PROGRAM PRG_CML_ValidationAsConfirmation
VAR

	rtrigNewOuterArrived				: R_TRIG;
	bNewOuterIsProccesing				: BOOL;
	tonValidationTimout					: TON;
	tofValidationTimout					: TOF;
	ftrigValidationTimout				: F_TRIG;
	bValidationTimeout					: BOOL;
	bValidationTimeoutReset				: BOOL;
	fbTooCloseCounter					: CTU;
	fbTimeoutCounter					: CTU;
	nCountTimeout					: WORD;
	nCountTooClose					: WORD;

	fbMasterListCamera				: FB_SCANNER_CameraSelect;
	(*stMasterListCameraOptions		: ST_SCANNER_Options := (eScannerType := E_MV_420_FULL, nImageBuffer := 1, nExpectedResp := 2);*)

	fbOuterValidationEvaluation		: FB_SCANNER_Evaluation;
	fbCheckForDuplicateMasterList	: FB_OUTER_CheckDuplicateStatus;

	rtrigOuterCameraDone				: R_TRIG;
	bOuterCameraDone				: BOOL;
	bDataReadyForValidation			: BOOL;
	bQAReject								: BOOL;

	sLastImageLableString				: T_OUTER_Barcode;

	fbPerformance							: FB_Interval;
	fbMoveOuterData						: FB_OUTER_MoveOuterStatus;
	fbCompleteDataFromConfirmation	: FB_OUTER_CompleteDataFromDB_SingleCam;
	fbMETSValidateOuterForReject			: FB_OUTER_ValidateOuterForReject;
	tofValidateOuterDoneForHMI			: TOF;
	fbMasterListUpdate					: FB_OUTER_MasterListUpdate;

	fbOuterLevelCounter				: FB_KPI_OuterLevelCounter;

	stLastOuterCompleted				: ST_OUTER_Status;
	sLastReadOuterBarcode			: T_OUTER_Barcode;
	sLastReadConfPackCode1			: T_PACK_Barcode;
	nOutersCompleted					: UDINT;
	bDoneInfo							: BOOL;
	rsTwoOutersOnRejectConv		: RS;
	bTwoOutersOnRejectConv			: BOOL;
	bCMLBiuldBackRejectActive		: BOOL;

	rtrigSetOuterValidationOK			: R_TRIG;
	rtrigSetOuterValidationNOK		: R_TRIG;
	rtrigResetValidationStatus			: R_TRIG;

	rsOuterRejectStation 				: RS;

	sRejectCode						: STRING(255);
	fbArchiveInvalidOuters			: FB_OUTER_ArchiveInvalidOuters;
	aReasonForReject					: ARRAY[0..50] OF STRING(255);
	bClearList							: BOOL;

	fbOuterProduced					: FB_KPI_GenericEfficiency;
	fbOuterInspection					: FB_KPI_OutersEfficiency;

	fbQARejectCounter				: FB_CTU32;
	fbOuterValidationIndexOK			: FB_CTU32;

	ctuConsecutiveOuterRejects		: CTU;
	nActualCount						: WORD;
END_VAR
VAR // added by the converter: edge detectors and wires of the graphical bodies
    _w1, _w2 : BOOL;
END_VAR

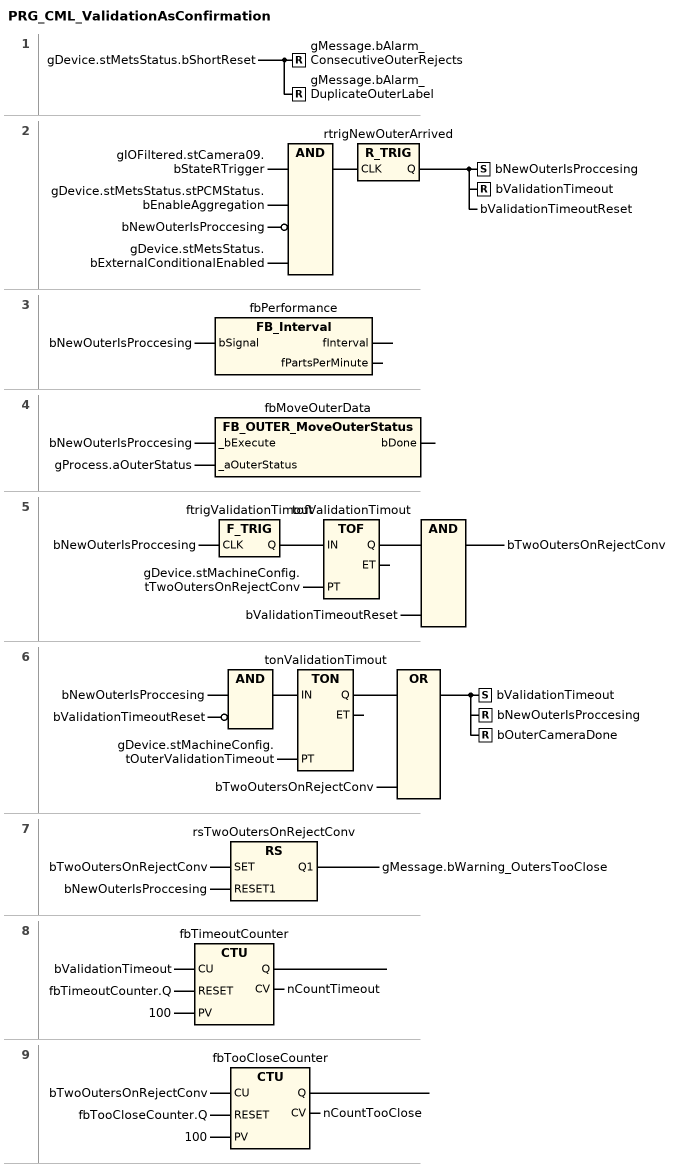
// NETWORK 1
gMessage.bAlarm_ConsecutiveOuterRejects R= gDevice.stMetsStatus.bShortReset;
gMessage.bAlarm_DuplicateOuterLabel R= gDevice.stMetsStatus.bShortReset;

// NETWORK 2
rtrigNewOuterArrived(CLK := gIOFiltered.stCamera09.bStateRTrigger AND gDevice.stMetsStatus.stPCMStatus.bEnableAggregation AND NOT bNewOuterIsProccesing AND gDevice.stMetsStatus.bExternalConditionalEnabled); // R_TRIG
bNewOuterIsProccesing S= rtrigNewOuterArrived.Q;
bValidationTimeout R= rtrigNewOuterArrived.Q;
bValidationTimeoutReset := rtrigNewOuterArrived.Q;

// NETWORK 3
fbPerformance(bSignal := bNewOuterIsProccesing); // FB_Interval

// NETWORK 4
fbMoveOuterData(_bExecute := bNewOuterIsProccesing, _aOuterStatus := gProcess.aOuterStatus); // FB_OUTER_MoveOuterStatus

// NETWORK 5
ftrigValidationTimout(CLK := bNewOuterIsProccesing); // F_TRIG
tofValidationTimout(IN := ftrigValidationTimout.Q, PT := gDevice.stMachineConfig.tTwoOutersOnRejectConv); // TOF
bTwoOutersOnRejectConv := tofValidationTimout.Q AND bValidationTimeoutReset;

// NETWORK 6
tonValidationTimout(IN := bNewOuterIsProccesing AND NOT bValidationTimeoutReset, PT := gDevice.stMachineConfig.tOuterValidationTimeout); // TON
_w1 := tonValidationTimout.Q OR bTwoOutersOnRejectConv;
bValidationTimeout S= _w1;
bNewOuterIsProccesing R= _w1;
bOuterCameraDone R= _w1;

// NETWORK 7
rsTwoOutersOnRejectConv(SET := bTwoOutersOnRejectConv, RESET1 := bNewOuterIsProccesing); // RS
gMessage.bWarning_OutersTooClose := rsTwoOutersOnRejectConv.Q1;

// NETWORK 8
fbTimeoutCounter(CU := bValidationTimeout, RESET := fbTimeoutCounter.Q, PV := 100, CV => nCountTimeout); // CTU

// NETWORK 9
fbTooCloseCounter(
    CU := bTwoOutersOnRejectConv,
    RESET := fbTooCloseCounter.Q,
    PV := 100,
    CV => nCountTooClose); // CTU

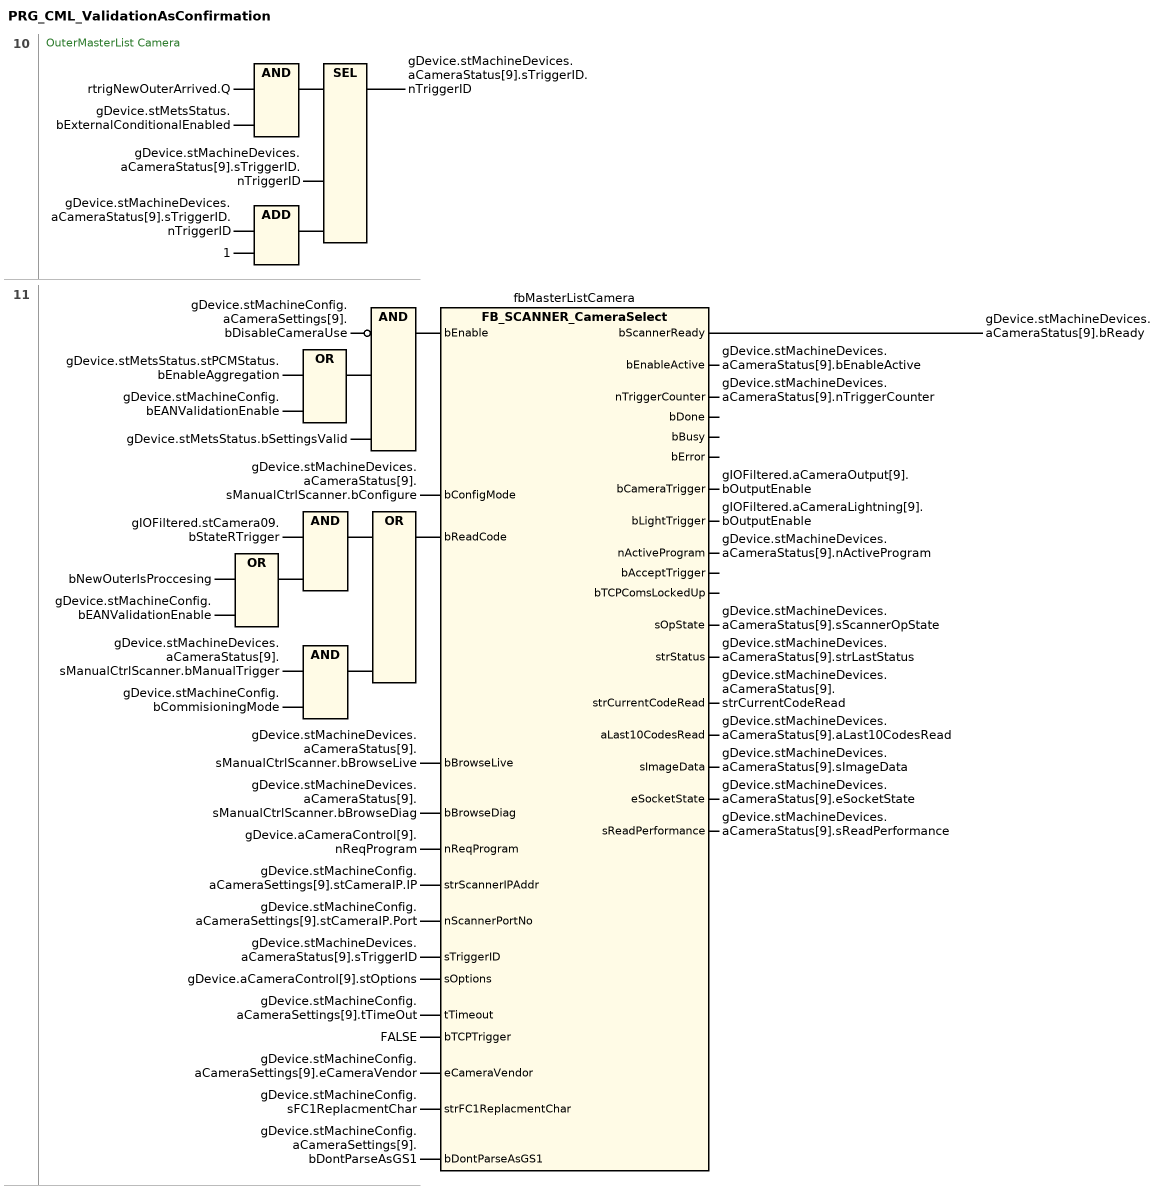
// NETWORK 10
// OuterMasterList Camera
gDevice.stMachineDevices.aCameraStatus[9].sTriggerID.nTriggerID := SEL(rtrigNewOuterArrived.Q AND gDevice.stMetsStatus.bExternalConditionalEnabled, gDevice.stMachineDevices.aCameraStatus[9].sTriggerID.nTriggerID, gDevice.stMachineDevices.aCameraStatus[9].sTriggerID.nTriggerID + 1);

// NETWORK 11
fbMasterListCamera(
    bEnable := NOT gDevice.stMachineConfig.aCameraSettings[9].bDisableCameraUse AND (gDevice.stMetsStatus.stPCMStatus.bEnableAggregation OR gDevice.stMachineConfig.bEANValidationEnable) AND gDevice.stMetsStatus.bSettingsValid,
    bConfigMode := gDevice.stMachineDevices.aCameraStatus[9].sManualCtrlScanner.bConfigure,
    bReadCode := gIOFiltered.stCamera09.bStateRTrigger AND (bNewOuterIsProccesing OR gDevice.stMachineConfig.bEANValidationEnable) OR gDevice.stMachineDevices.aCameraStatus[9].sManualCtrlScanner.bManualTrigger AND gDevice.stMachineConfig.bCommisioningMode,
    bBrowseLive := gDevice.stMachineDevices.aCameraStatus[9].sManualCtrlScanner.bBrowseLive,
    bBrowseDiag := gDevice.stMachineDevices.aCameraStatus[9].sManualCtrlScanner.bBrowseDiag,
    nReqProgram := gDevice.aCameraControl[9].nReqProgram,
    strScannerIPAddr := gDevice.stMachineConfig.aCameraSettings[9].stCameraIP.IP,
    nScannerPortNo := gDevice.stMachineConfig.aCameraSettings[9].stCameraIP.Port,
    sTriggerID := gDevice.stMachineDevices.aCameraStatus[9].sTriggerID,
    sOptions := gDevice.aCameraControl[9].stOptions,
    tTimeout := gDevice.stMachineConfig.aCameraSettings[9].tTimeOut,
    bTCPTrigger := FALSE,
    eCameraVendor := gDevice.stMachineConfig.aCameraSettings[9].eCameraVendor,
    strFC1ReplacmentChar := gDevice.stMachineConfig.sFC1ReplacmentChar,
    bDontParseAsGS1 := gDevice.stMachineConfig.aCameraSettings[9].bDontParseAsGS1,
    bEnableActive => gDevice.stMachineDevices.aCameraStatus[9].bEnableActive,
    nTriggerCounter => gDevice.stMachineDevices.aCameraStatus[9].nTriggerCounter,
    bCameraTrigger => gIOFiltered.aCameraOutput[9].bOutputEnable,
    bLightTrigger => gIOFiltered.aCameraLightning[9].bOutputEnable,
    nActiveProgram => gDevice.stMachineDevices.aCameraStatus[9].nActiveProgram,
    sOpState => gDevice.stMachineDevices.aCameraStatus[9].sScannerOpState,
    strStatus => gDevice.stMachineDevices.aCameraStatus[9].strLastStatus,
    strCurrentCodeRead => gDevice.stMachineDevices.aCameraStatus[9].strCurrentCodeRead,
    aLast10CodesRead => gDevice.stMachineDevices.aCameraStatus[9].aLast10CodesRead,
    sImageData => gDevice.stMachineDevices.aCameraStatus[9].sImageData,
    eSocketState => gDevice.stMachineDevices.aCameraStatus[9].eSocketState,
    sReadPerformance => gDevice.stMachineDevices.aCameraStatus[9].sReadPerformance); // FB_SCANNER_CameraSelect
gDevice.stMachineDevices.aCameraStatus[9].bReady := fbMasterListCamera.bScannerReady;

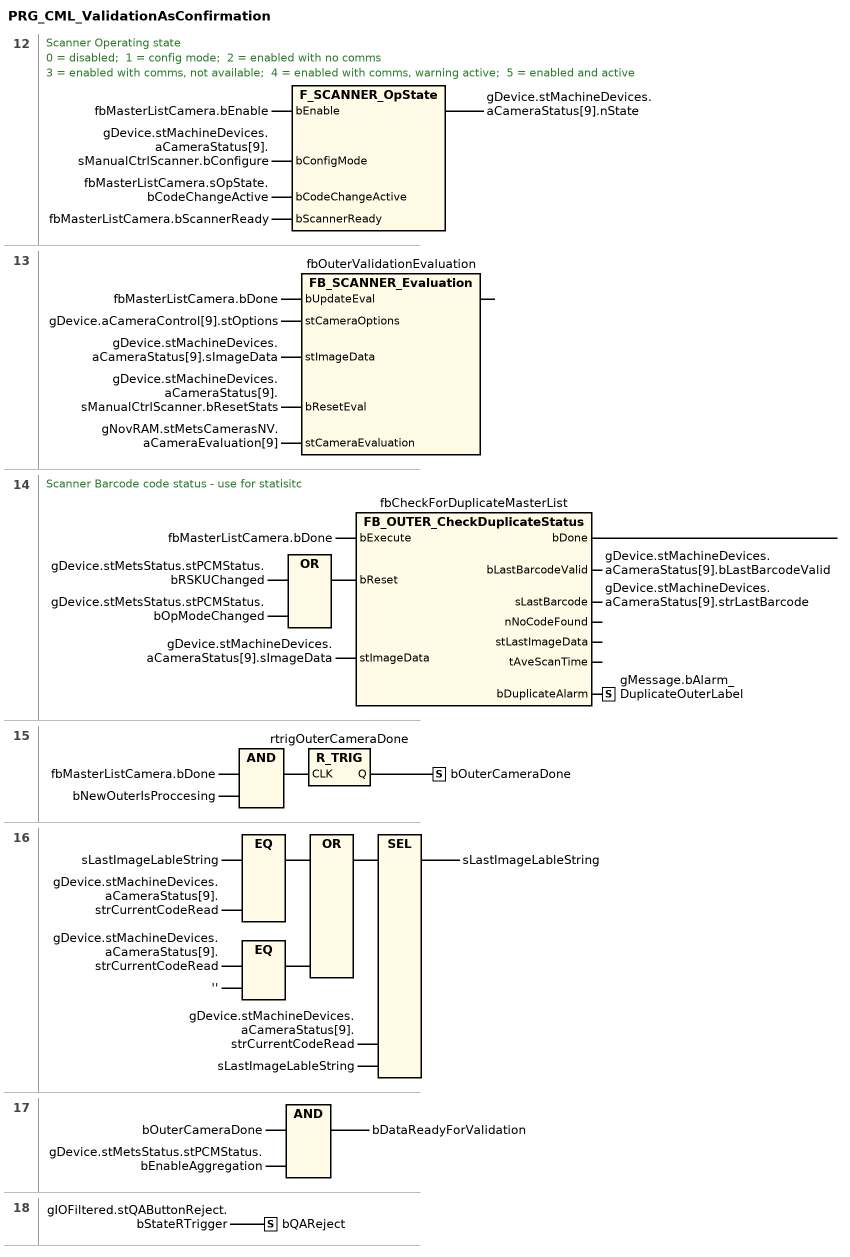
// NETWORK 12
// 					Scanner Operating state
// 0 = disabled;  1 = config mode;  2 = enabled with no comms
// 3 = enabled with comms, not available;  4 = enabled with comms, warning active;  5 = enabled and active
//
gDevice.stMachineDevices.aCameraStatus[9].nState := F_SCANNER_OpState(bEnable := fbMasterListCamera.bEnable, bConfigMode := gDevice.stMachineDevices.aCameraStatus[9].sManualCtrlScanner.bConfigure, bCodeChangeActive := fbMasterListCamera.sOpState.bCodeChangeActive, bScannerReady := fbMasterListCamera.bScannerReady);

// NETWORK 13
fbOuterValidationEvaluation(
    bUpdateEval := fbMasterListCamera.bDone,
    stCameraOptions := gDevice.aCameraControl[9].stOptions,
    stImageData := gDevice.stMachineDevices.aCameraStatus[9].sImageData,
    bResetEval := gDevice.stMachineDevices.aCameraStatus[9].sManualCtrlScanner.bResetStats,
    stCameraEvaluation := gNovRAM.stMetsCamerasNV.aCameraEvaluation[9]); // FB_SCANNER_Evaluation

// NETWORK 14
// Scanner Barcode code status - use for statisitc
fbCheckForDuplicateMasterList(
    bExecute := fbMasterListCamera.bDone,
    bReset := gDevice.stMetsStatus.stPCMStatus.bRSKUChanged OR gDevice.stMetsStatus.stPCMStatus.bOpModeChanged,
    stImageData := gDevice.stMachineDevices.aCameraStatus[9].sImageData,
    bLastBarcodeValid => gDevice.stMachineDevices.aCameraStatus[9].bLastBarcodeValid,
    sLastBarcode => gDevice.stMachineDevices.aCameraStatus[9].strLastBarcode); // FB_OUTER_CheckDuplicateStatus
gMessage.bAlarm_DuplicateOuterLabel S= fbCheckForDuplicateMasterList.bDuplicateAlarm;

// NETWORK 15
rtrigOuterCameraDone(CLK := fbMasterListCamera.bDone AND bNewOuterIsProccesing); // R_TRIG
bOuterCameraDone S= rtrigOuterCameraDone.Q;

// NETWORK 16
sLastImageLableString := SEL(sLastImageLableString = gDevice.stMachineDevices.aCameraStatus[9].strCurrentCodeRead OR gDevice.stMachineDevices.aCameraStatus[9].strCurrentCodeRead = '', gDevice.stMachineDevices.aCameraStatus[9].strCurrentCodeRead, sLastImageLableString);

// NETWORK 17
bDataReadyForValidation := bOuterCameraDone AND gDevice.stMetsStatus.stPCMStatus.bEnableAggregation;

// NETWORK 18
bQAReject S= gIOFiltered.stQAButtonReject.bStateRTrigger;

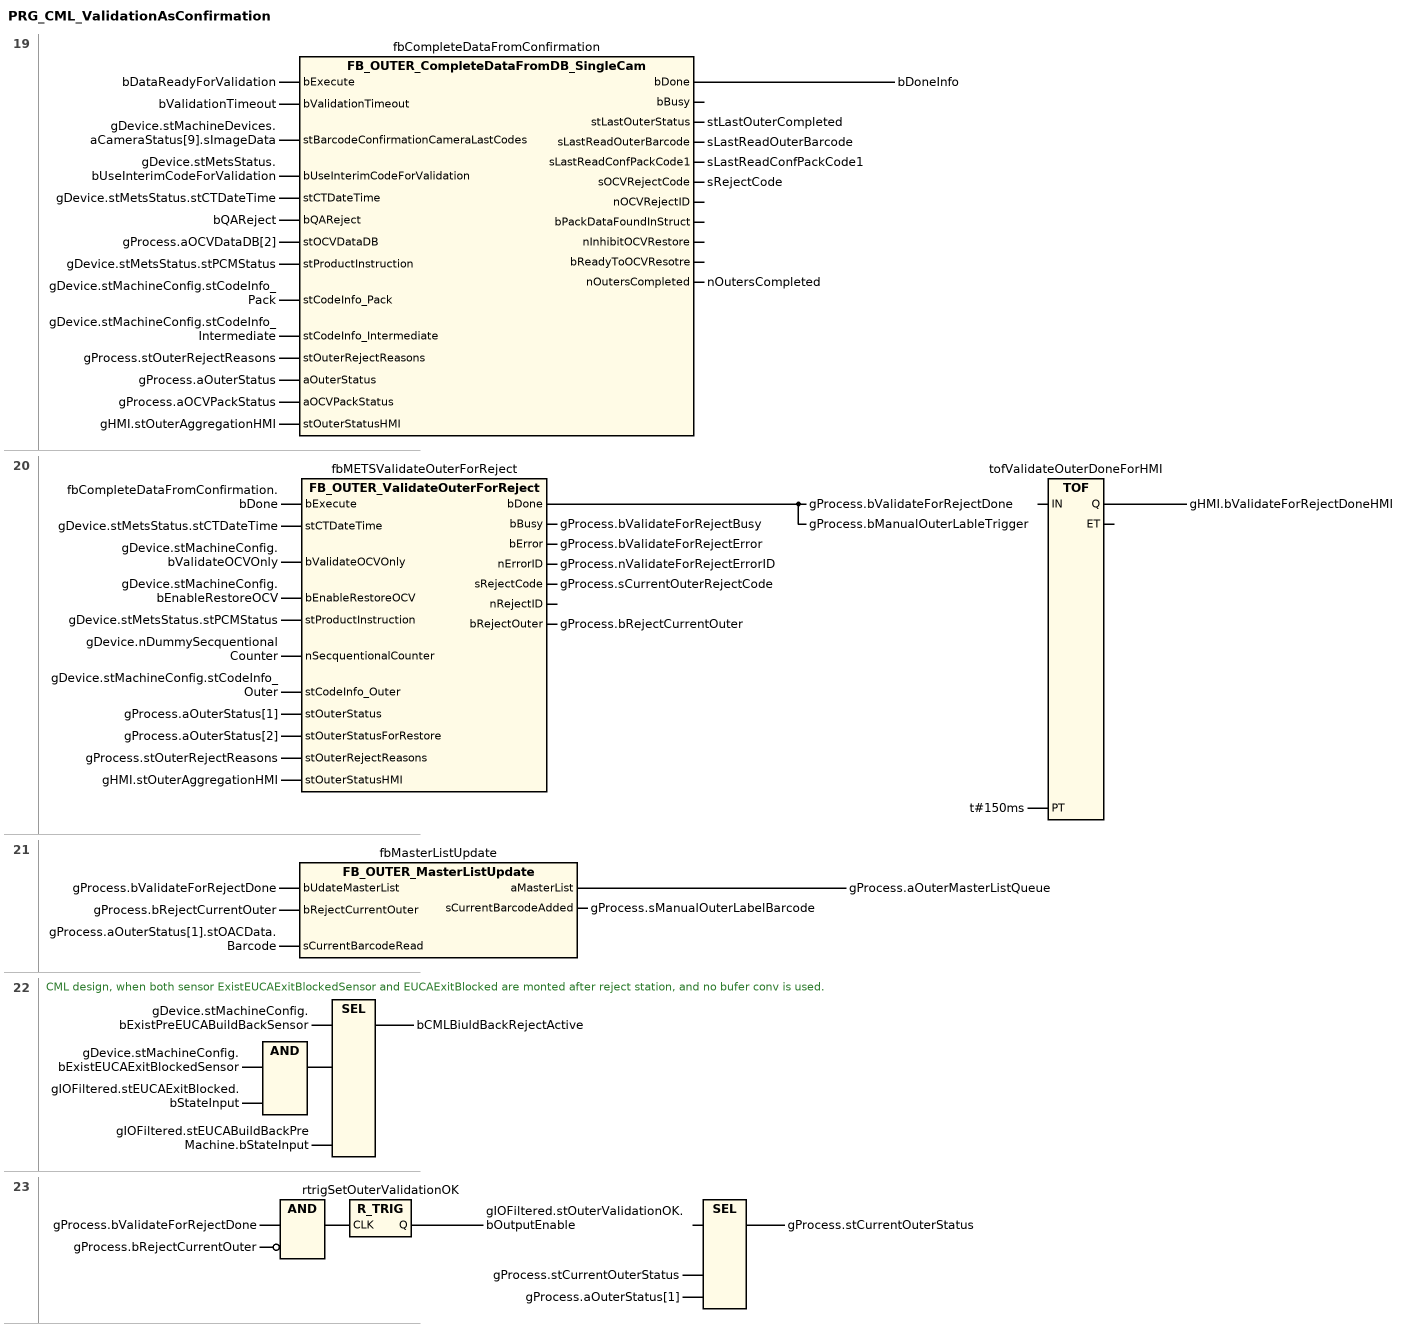
// NETWORK 19
fbCompleteDataFromConfirmation(
    bExecute := bDataReadyForValidation,
    bValidationTimeout := bValidationTimeout,
    stBarcodeConfirmationCameraLastCodes := gDevice.stMachineDevices.aCameraStatus[9].sImageData,
    bUseInterimCodeForValidation := gDevice.stMetsStatus.bUseInterimCodeForValidation,
    stCTDateTime := gDevice.stMetsStatus.stCTDateTime,
    bQAReject := bQAReject,
    stOCVDataDB := gProcess.aOCVDataDB[2],
    stProductInstruction := gDevice.stMetsStatus.stPCMStatus,
    stCodeInfo_Pack := gDevice.stMachineConfig.stCodeInfo_Pack,
    stCodeInfo_Intermediate := gDevice.stMachineConfig.stCodeInfo_Intermediate,
    stOuterRejectReasons := gProcess.stOuterRejectReasons,
    aOuterStatus := gProcess.aOuterStatus,
    aOCVPackStatus := gProcess.aOCVPackStatus,
    stOuterStatusHMI := gHMI.stOuterAggregationHMI,
    stLastOuterStatus => stLastOuterCompleted,
    sLastReadOuterBarcode => sLastReadOuterBarcode,
    sLastReadConfPackCode1 => sLastReadConfPackCode1,
    sOCVRejectCode => sRejectCode,
    nOutersCompleted => nOutersCompleted); // FB_OUTER_CompleteDataFromDB_SingleCam
bDoneInfo := fbCompleteDataFromConfirmation.bDone;

// NETWORK 20
fbMETSValidateOuterForReject(
    bExecute := fbCompleteDataFromConfirmation.bDone,
    stCTDateTime := gDevice.stMetsStatus.stCTDateTime,
    bValidateOCVOnly := gDevice.stMachineConfig.bValidateOCVOnly,
    bEnableRestoreOCV := gDevice.stMachineConfig.bEnableRestoreOCV,
    stProductInstruction := gDevice.stMetsStatus.stPCMStatus,
    nSecquentionalCounter := gDevice.nDummySecquentionalCounter,
    stCodeInfo_Outer := gDevice.stMachineConfig.stCodeInfo_Outer,
    stOuterStatus := gProcess.aOuterStatus[1],
    stOuterStatusForRestore := gProcess.aOuterStatus[2],
    stOuterRejectReasons := gProcess.stOuterRejectReasons,
    stOuterStatusHMI := gHMI.stOuterAggregationHMI,
    bBusy => gProcess.bValidateForRejectBusy,
    bError => gProcess.bValidateForRejectError,
    nErrorID => gProcess.nValidateForRejectErrorID,
    sRejectCode => gProcess.sCurrentOuterRejectCode,
    bRejectOuter => gProcess.bRejectCurrentOuter); // FB_OUTER_ValidateOuterForReject
gProcess.bValidateForRejectDone := fbMETSValidateOuterForReject.bDone;
gProcess.bManualOuterLableTrigger := fbMETSValidateOuterForReject.bDone;
tofValidateOuterDoneForHMI(IN := fbMETSValidateOuterForReject.bDone, PT := t#150ms); // TOF
gHMI.bValidateForRejectDoneHMI := tofValidateOuterDoneForHMI.Q;

// NETWORK 21
fbMasterListUpdate(
    bUdateMasterList := gProcess.bValidateForRejectDone,
    bRejectCurrentOuter := gProcess.bRejectCurrentOuter,
    sCurrentBarcodeRead := gProcess.aOuterStatus[1].stOACData.Barcode,
    sCurrentBarcodeAdded => gProcess.sManualOuterLabelBarcode); // FB_OUTER_MasterListUpdate
gProcess.aOuterMasterListQueue := fbMasterListUpdate.aMasterList;

// NETWORK 22
// CML design, when both sensor ExistEUCAExitBlockedSensor and EUCAExitBlocked are monted after reject station, and no bufer conv is used.
bCMLBiuldBackRejectActive := SEL(gDevice.stMachineConfig.bExistPreEUCABuildBackSensor, gDevice.stMachineConfig.bExistEUCAExitBlockedSensor AND gIOFiltered.stEUCAExitBlocked.bStateInput, gIOFiltered.stEUCABuildBackPreMachine.bStateInput);

// NETWORK 23
rtrigSetOuterValidationOK(CLK := gProcess.bValidateForRejectDone AND NOT gProcess.bRejectCurrentOuter); // R_TRIG
gIOFiltered.stOuterValidationOK.bOutputEnable := rtrigSetOuterValidationOK.Q;
gProcess.stCurrentOuterStatus := SEL(rtrigSetOuterValidationOK.Q, gProcess.stCurrentOuterStatus, gProcess.aOuterStatus[1]);

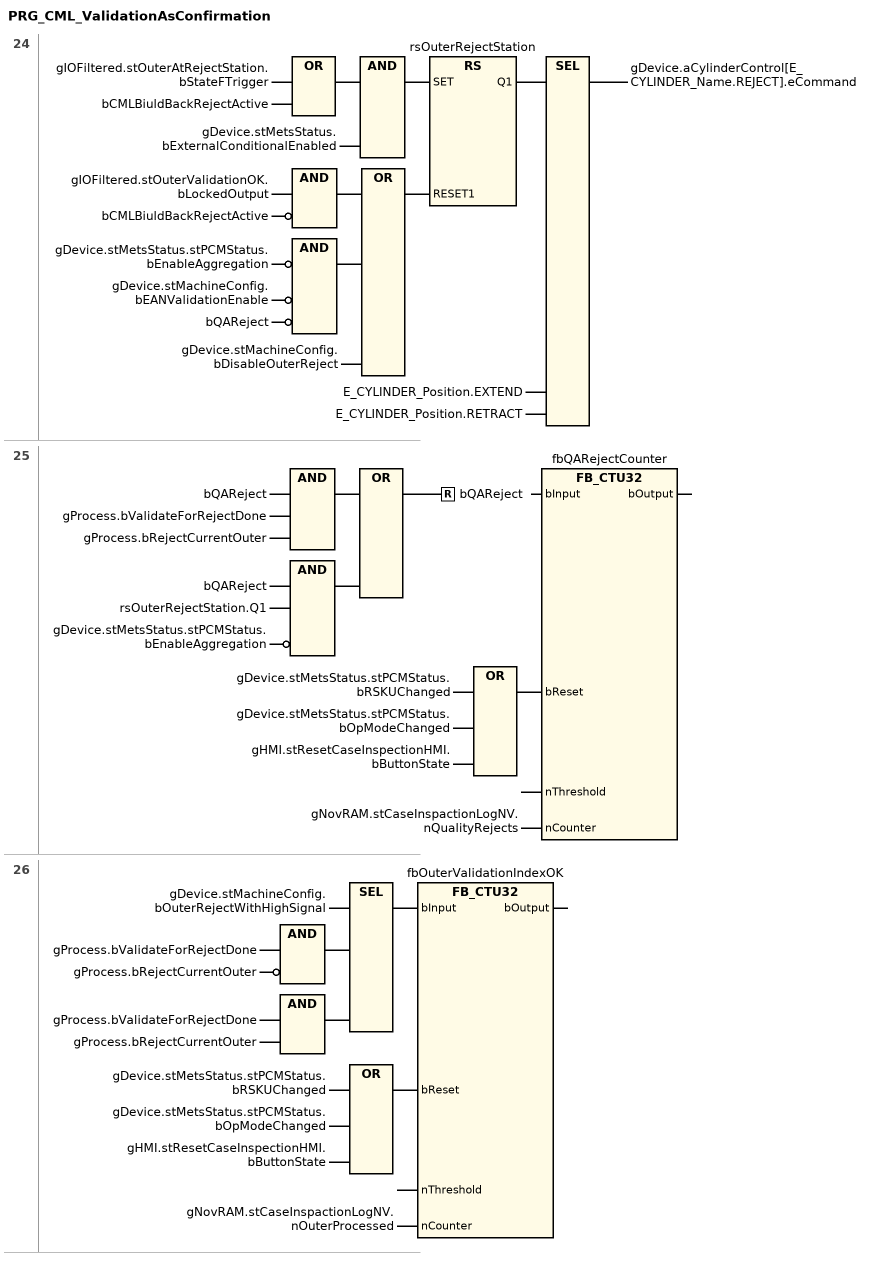
// NETWORK 24
rsOuterRejectStation(SET := (gIOFiltered.stOuterAtRejectStation.bStateFTrigger OR bCMLBiuldBackRejectActive) AND gDevice.stMetsStatus.bExternalConditionalEnabled, RESET1 := gIOFiltered.stOuterValidationOK.bLockedOutput AND NOT bCMLBiuldBackRejectActive OR NOT gDevice.stMetsStatus.stPCMStatus.bEnableAggregation AND NOT gDevice.stMachineConfig.bEANValidationEnable AND NOT bQAReject OR gDevice.stMachineConfig.bDisableOuterReject); // RS
gDevice.aCylinderControl[E_CYLINDER_Name.REJECT].eCommand := SEL(rsOuterRejectStation.Q1, E_CYLINDER_Position.EXTEND, E_CYLINDER_Position.RETRACT);

// NETWORK 25
_w2 := bQAReject AND gProcess.bValidateForRejectDone AND gProcess.bRejectCurrentOuter OR bQAReject AND rsOuterRejectStation.Q1 AND NOT gDevice.stMetsStatus.stPCMStatus.bEnableAggregation;
bQAReject R= _w2;
fbQARejectCounter(
    bInput := _w2,
    bReset := gDevice.stMetsStatus.stPCMStatus.bRSKUChanged OR gDevice.stMetsStatus.stPCMStatus.bOpModeChanged OR gHMI.stResetCaseInspectionHMI.bButtonState,
    nCounter := gNovRAM.stCaseInspactionLogNV.nQualityRejects); // FB_CTU32

// NETWORK 26
fbOuterValidationIndexOK(
    bInput := SEL(gDevice.stMachineConfig.bOuterRejectWithHighSignal, gProcess.bValidateForRejectDone AND NOT gProcess.bRejectCurrentOuter, gProcess.bValidateForRejectDone AND gProcess.bRejectCurrentOuter),
    bReset := gDevice.stMetsStatus.stPCMStatus.bRSKUChanged OR gDevice.stMetsStatus.stPCMStatus.bOpModeChanged OR gHMI.stResetCaseInspectionHMI.bButtonState,
    nCounter := gNovRAM.stCaseInspactionLogNV.nOuterProcessed); // FB_CTU32

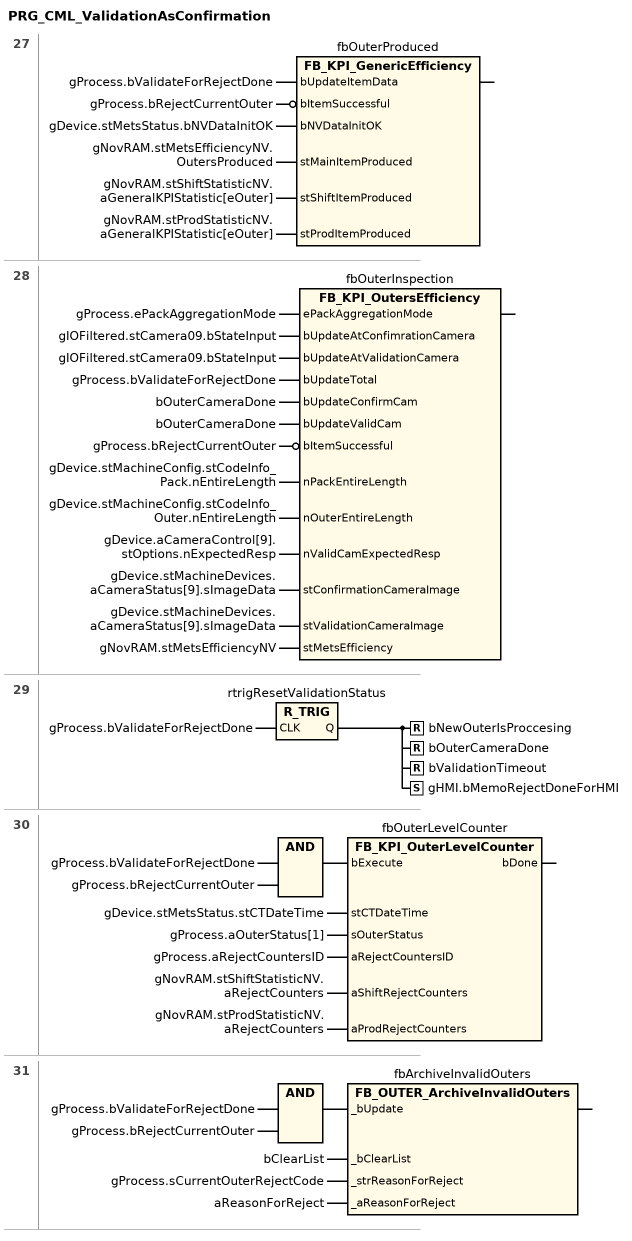
// NETWORK 27
fbOuterProduced(
    bUpdateItemData := gProcess.bValidateForRejectDone,
    bItemSuccessful := NOT gProcess.bRejectCurrentOuter,
    bNVDataInitOK := gDevice.stMetsStatus.bNVDataInitOK,
    stMainItemProduced := gNovRAM.stMetsEfficiencyNV.OutersProduced,
    stShiftItemProduced := gNovRAM.stShiftStatisticNV.aGeneralKPIStatistic[eOuter],
    stProdItemProduced := gNovRAM.stProdStatisticNV.aGeneralKPIStatistic[eOuter]); // FB_KPI_GenericEfficiency

// NETWORK 28
fbOuterInspection(
    ePackAggregationMode := gProcess.ePackAggregationMode,
    bUpdateAtConfimrationCamera := gIOFiltered.stCamera09.bStateInput,
    bUpdateAtValidationCamera := gIOFiltered.stCamera09.bStateInput,
    bUpdateTotal := gProcess.bValidateForRejectDone,
    bUpdateConfirmCam := bOuterCameraDone,
    bUpdateValidCam := bOuterCameraDone,
    bItemSuccessful := NOT gProcess.bRejectCurrentOuter,
    nPackEntireLength := gDevice.stMachineConfig.stCodeInfo_Pack.nEntireLength,
    nOuterEntireLength := gDevice.stMachineConfig.stCodeInfo_Outer.nEntireLength,
    nValidCamExpectedResp := gDevice.aCameraControl[9].stOptions.nExpectedResp,
    stConfirmationCameraImage := gDevice.stMachineDevices.aCameraStatus[9].sImageData,
    stValidationCameraImage := gDevice.stMachineDevices.aCameraStatus[9].sImageData,
    stMetsEfficiency := gNovRAM.stMetsEfficiencyNV); // FB_KPI_OutersEfficiency

// NETWORK 29
rtrigResetValidationStatus(CLK := gProcess.bValidateForRejectDone); // R_TRIG
bNewOuterIsProccesing R= rtrigResetValidationStatus.Q;
bOuterCameraDone R= rtrigResetValidationStatus.Q;
bValidationTimeout R= rtrigResetValidationStatus.Q;
gHMI.bMemoRejectDoneForHMI S= rtrigResetValidationStatus.Q;

// NETWORK 30
fbOuterLevelCounter(
    bExecute := gProcess.bValidateForRejectDone AND gProcess.bRejectCurrentOuter,
    stCTDateTime := gDevice.stMetsStatus.stCTDateTime,
    sOuterStatus := gProcess.aOuterStatus[1],
    aRejectCountersID := gProcess.aRejectCountersID,
    aShiftRejectCounters := gNovRAM.stShiftStatisticNV.aRejectCounters,
    aProdRejectCounters := gNovRAM.stProdStatisticNV.aRejectCounters); // FB_KPI_OuterLevelCounter

// NETWORK 31
fbArchiveInvalidOuters(
    _bUpdate := gProcess.bValidateForRejectDone AND gProcess.bRejectCurrentOuter,
    _bClearList := bClearList,
    _strReasonForReject := gProcess.sCurrentOuterRejectCode,
    _aReasonForReject := aReasonForReject); // FB_OUTER_ArchiveInvalidOuters

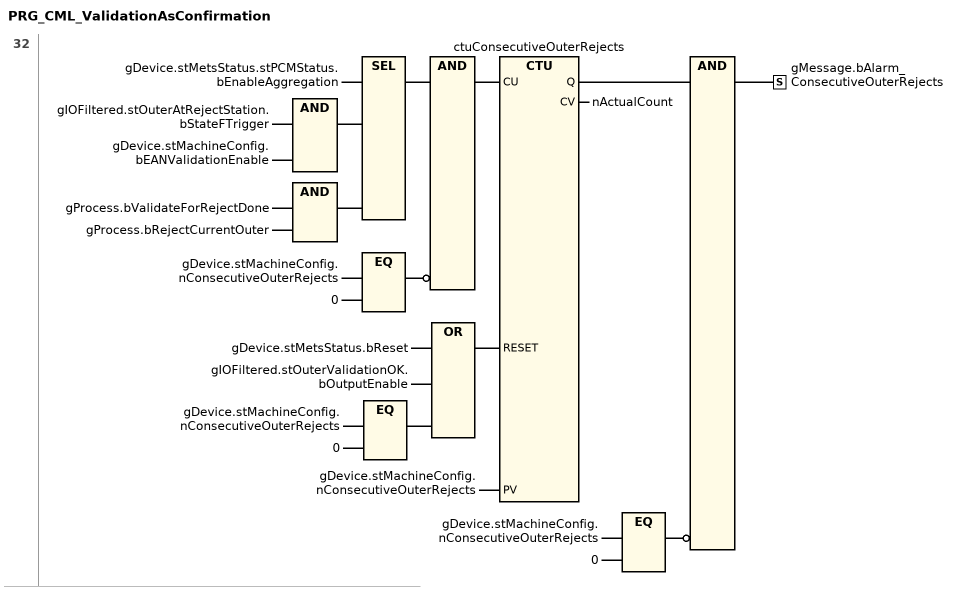
// NETWORK 32
ctuConsecutiveOuterRejects(
    CU := SEL(gDevice.stMetsStatus.stPCMStatus.bEnableAggregation, gIOFiltered.stOuterAtRejectStation.bStateFTrigger AND gDevice.stMachineConfig.bEANValidationEnable, gProcess.bValidateForRejectDone AND gProcess.bRejectCurrentOuter) AND NOT (gDevice.stMachineConfig.nConsecutiveOuterRejects = 0),
    RESET := gDevice.stMetsStatus.bReset OR gIOFiltered.stOuterValidationOK.bOutputEnable OR gDevice.stMachineConfig.nConsecutiveOuterRejects = 0,
    PV := gDevice.stMachineConfig.nConsecutiveOuterRejects,
    CV => nActualCount); // CTU
gMessage.bAlarm_ConsecutiveOuterRejects S= ctuConsecutiveOuterRejects.Q AND NOT (gDevice.stMachineConfig.nConsecutiveOuterRejects = 0);

END_PROGRAM

(* stored: Version 1.1.0.1
   POU PRG_CML_ValidationAsConfirmation: Id {e1c1291d-50ed-4b30-b3eb-05db38927f79}, SpecialFunc None *)
